// TIA Portal project "EqualAging" (V15)

(* hardware
DEVICE "S7-1200 station_1"  S7-1200 Station
   slot 0: "Rack_0"  S7-1200 Rack  Rack  V1.0
   slot 1: "PLC_1"  CPU 1214C DC/DC/DC  6ES7 214-1AG40-0XB0  V4.2
*)

// ===== PLC "PLC_1"  CPU 1214C DC/DC/DC =====

VAR_GLOBAL   // PLC tag table "Default tag table"
   "Tag_2" AT %Q0.0 : Bool;
   "Tag_3" AT %M1.0 : Bool;
   "Tag_4" AT %M1.1 : Bool;
   "Tag_5" AT %M1.2 : Bool;
   "Tag_6" AT %M1.3 : Bool;
   "Tag_7" AT %M1.4 : Bool;
   "Tag_8" AT %M1.5 : Bool;
   "Tag_9" AT %M1.6 : Bool;
   "Tag_10" AT %MW20 : Int;
   "Tag_11" AT %MD10 : Time;
   "Tag_12" AT %MD11 : Time;
   "Tag_13" AT %MD16 : Time;
   "Clock_Byte" AT %MB0 : Byte;
   "Clock_10Hz" AT %M0.0 : Bool;
   "Clock_5Hz" AT %M0.1 : Bool;
   "Clock_2.5Hz" AT %M0.2 : Bool;
   "Clock_2Hz" AT %M0.3 : Bool;
   "Clock_1.25Hz" AT %M0.4 : Bool;
   "Clock_1Hz" AT %M0.5 : Bool;
   "Clock_0.625Hz" AT %M0.6 : Bool;
   "Clock_0.5Hz" AT %M0.7 : Bool;
   "Tag_1" AT %M10.0 : Bool;
   "Tag_14" AT %M10.1 : Bool;
   "Tag_15" AT %M10.2 : Bool;
   "Tag_16" AT %M10.3 : Bool;
   "Tag_17" AT %M10.4 : Bool;
END_VAR

DATA_BLOCK "EqualAging_DB"   // DB1
{ S7_Optimized_Access := 'TRUE' }
VERSION : 0.1
// stored: InstanceOfName EqualAging
"EqualAging"
BEGIN
END_DATA_BLOCK

FUNCTION_BLOCK "EqualAging"   // FB1, SCL
{ S7_Optimized_Access := 'TRUE' }
VERSION : 0.1
   VAR_INPUT
      i_SystemEnable : Bool;   // Sistemi genel aç/kapat anahtarı
      i_ResetAlarms : Bool;   // Arıza ve saatleri resetler
      i_Clock_1Hz : Bool;   // Saat sayımı için 1 saniyelik darbe
      i_SetMotorCount : Int;   // Çalıştırılmak istenen motor sayısı
      i_StageDelayTime : Time;   // Motorlar arası devreye girme süresi
      i_RotationInterval : Time;   // Motor değişim süresi
      i_M1_Ready : Bool;   // 1. motor hazır/sağlam
      i_M2_Ready : Bool;   // 2. motor hazır/sağlam
      i_M3_Ready : Bool;   // 3. motor hazır/sağlam
      i_M4_Ready : Bool;   // 4. motor hazır/sağlam
      i_M5_Ready : Bool;   // 5. motor hazır/sağlam
   END_VAR
   VAR_OUTPUT
      q_M1_Start : Bool;   // 1. motor çalıştır komutu
      q_M2_Start : Bool;   // 2. motor çalıştır komutu
      q_M3_Start : Bool;   // 3. motor çalıştır komutu
      q_M4_Start : Bool;   // 4. motor çalıştır komutu
      q_M5_Start : Bool;   // 5. motor çalıştır komutu
      q_M1_Hours : Real;   // 1. motor çalışma saati
      q_M2_Hours : Real;   // 2. motor çalışma saati
      q_M3_Hours : Real;   // 3. motor çalışma saati
      q_M4_Hours : Real;   // 4. motor çalışma saati
      q_M5_Hours : Real;   // 5. motor çalışma saati
      q_ActiveCount : Int;   // aktif çalışan motor sayısı
      q_RotationTrigger : Bool;
      q_InsufficientCap : Bool;   // Kapasite yetersiz uyarısı
   END_VAR
   VAR
      stat_RTrig : R_TRIG;   // Saat darbesini yakalamak için
   END_VAR
   VAR RETAIN
      stat_RunSecs : Array[0..5] of DInt;   // motorların toplam süresi
   END_VAR
   VAR
      stat_RotationTimer : TON_TIME;
      stat_CmdStart : Array[0..5] of Bool;   // Çıkışları yönetmek için iç hafıza
      stat_StageTimer : TON_TIME;
   END_VAR
   VAR_TEMP
      temp_i : Int;
      temp_k : Int;
      temp_AvailQty : Int;
      temp_RunQty_1 : Int;
      temp_MinTime : DInt;
      temp_MaxTime : DInt;
      temp_BestStart : Int;
      temp_BestStop : Int;
      temp_Ready : Array[0..5] of Bool;
      temp_SafeSet : Int;
      temp_RunQty : Int;
   END_VAR
BEGIN


   // 1. GİRİŞLERİ DİZİYE AKTARMA (MAPPING)
   #temp_Ready[1] := #i_M1_Ready;
   #temp_Ready[2] := #i_M2_Ready;
   #temp_Ready[3] := #i_M3_Ready;
   #temp_Ready[4] := #i_M4_Ready;
   #temp_Ready[5] := #i_M5_Ready;

   // Saat Palsini Yakala
   #stat_RTrig(CLK := #i_Clock_1Hz);

   #temp_AvailQty := 0;
   #temp_RunQty := 0;

   FOR #temp_i := 1 TO 5 DO
       // Saat Sayacı 
       IF #stat_CmdStart[#temp_i] AND #stat_RTrig.Q THEN
           #stat_RunSecs[#temp_i] := #stat_RunSecs[#temp_i] + 1;
       END_IF;

       // Reset İşlemi 
       IF #i_ResetAlarms THEN
           #stat_RunSecs[#temp_i] := 0;
       END_IF;

       // Hazır Değilse Start'ı Kes
       IF NOT #temp_Ready[#temp_i] THEN
           #stat_CmdStart[#temp_i] := FALSE;
       ELSE
           // Hazırsa "Sağlam" sayısına ekle
           #temp_AvailQty := #temp_AvailQty + 1;
       END_IF;

       // Çalışanları Say 
       IF #stat_CmdStart[#temp_i] THEN
           #temp_RunQty := #temp_RunQty + 1;
       END_IF;
   END_FOR;

   // Çıkışa Aktar
   #q_ActiveCount := #temp_RunQty;

   // Kapasite Kontrolü
   IF #i_SetMotorCount > #temp_AvailQty THEN
       #q_InsufficientCap := TRUE;
       #temp_SafeSet := #temp_AvailQty;
   ELSE
       #q_InsufficientCap := FALSE;
       #temp_SafeSet := #i_SetMotorCount;
   END_IF;

   // --- ROTASYON ZAMANLAYICISI ---
   #stat_RotationTimer(IN := #i_SystemEnable AND
                       (#temp_RunQty = #temp_SafeSet) AND
                       (#temp_RunQty > 0) AND
                       (#temp_AvailQty > #temp_SafeSet),
                       PT := #i_RotationInterval);

   #q_RotationTrigger := #stat_RotationTimer.Q;

   IF #stat_RotationTimer.Q THEN
       #temp_MaxTime := -1;
       #temp_BestStop := 0;

       FOR #temp_k := 1 TO 5 DO
           IF #stat_CmdStart[#temp_k] THEN
               IF #stat_RunSecs[#temp_k] > #temp_MaxTime THEN
                   #temp_MaxTime := #stat_RunSecs[#temp_k];
                   #temp_BestStop := #temp_k;
               END_IF;
           END_IF;
       END_FOR;

       IF #temp_BestStop > 0 THEN
           #stat_CmdStart[#temp_BestStop] := FALSE;
       END_IF;
   END_IF;

   // --- GEÇİŞ ZAMANLAYICISI ---
   #stat_StageTimer(IN := (#temp_RunQty <> #temp_SafeSet) AND #i_SystemEnable,
                    PT := #i_StageDelayTime);

   IF #stat_StageTimer.Q AND #i_SystemEnable THEN

       // START VERME 
       IF #temp_RunQty < #temp_SafeSet THEN
           #temp_MinTime := 2147483647;
           #temp_BestStart := 0;

           FOR #temp_k := 1 TO 5 DO
               IF #temp_Ready[#temp_k] AND NOT #stat_CmdStart[#temp_k] THEN
                   IF #stat_RunSecs[#temp_k] < #temp_MinTime THEN
                       #temp_MinTime := #stat_RunSecs[#temp_k];
                       #temp_BestStart := #temp_k;
                   END_IF;
               END_IF;
           END_FOR;

           IF #temp_BestStart > 0 THEN
               #stat_CmdStart[#temp_BestStart] := TRUE;
           END_IF;

           // STOP VERME
       ELSIF #temp_RunQty > #temp_SafeSet THEN
           #temp_MaxTime := -1;
           #temp_BestStop := 0;

           FOR #temp_k := 1 TO 5 DO
               IF #stat_CmdStart[#temp_k] THEN
                   IF #stat_RunSecs[#temp_k] > #temp_MaxTime THEN
                       #temp_MaxTime := #stat_RunSecs[#temp_k];
                       #temp_BestStop := #temp_k;
                   END_IF;
               END_IF;
           END_FOR;

           IF #temp_BestStop > 0 THEN
               #stat_CmdStart[#temp_BestStop] := FALSE;
           END_IF;
       END_IF;
   END_IF;

   // Sistem Kapalıysa Hepsini Kes
   IF NOT #i_SystemEnable THEN
       FOR #temp_i := 1 TO 5 DO
           #stat_CmdStart[#temp_i] := FALSE;
       END_FOR;
   END_IF;

   // ÇIKIŞLARI AKTARMA
   #q_M1_Start := #stat_CmdStart[1];
   #q_M2_Start := #stat_CmdStart[2];
   #q_M3_Start := #stat_CmdStart[3];
   #q_M4_Start := #stat_CmdStart[4];
   #q_M5_Start := #stat_CmdStart[5];

   #q_M1_Hours := DINT_TO_REAL(#stat_RunSecs[1]) / 3600.0;
   #q_M2_Hours := DINT_TO_REAL(#stat_RunSecs[2]) / 3600.0;
   #q_M3_Hours := DINT_TO_REAL(#stat_RunSecs[3]) / 3600.0;
   #q_M4_Hours := DINT_TO_REAL(#stat_RunSecs[4]) / 3600.0;
   #q_M5_Hours := DINT_TO_REAL(#stat_RunSecs[5]) / 3600.0;
END_FUNCTION_BLOCK

ORGANIZATION_BLOCK "Main"   // OB1, LAD, ProgramCycle
TITLE = "Main Program Sweep (Cycle)"
{ S7_Optimized_Access := 'TRUE' }
VERSION : 0.1
   VAR_INPUT
      Initial_Call : Bool;   // Initial call of this OB
      Remanence : Bool;   // =True, if remanent data are available
   END_VAR
BEGIN

REGION Network 1
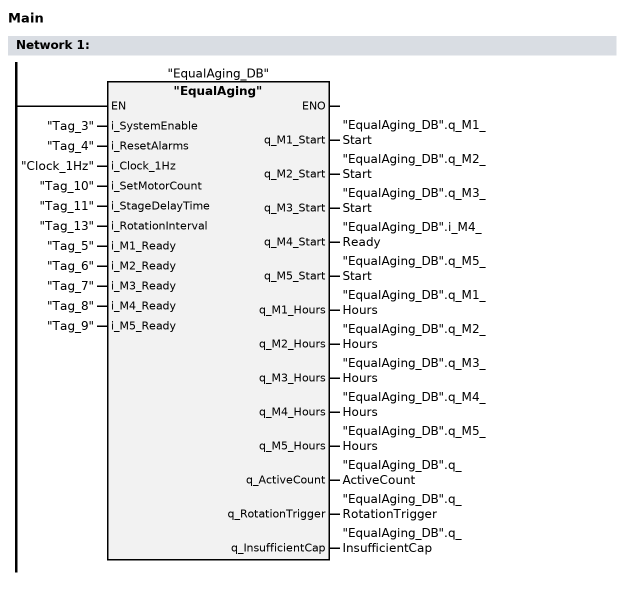
   RUNG wire#powerrail
      "EqualAging_DB"(i_SystemEnable := "Tag_3", i_ResetAlarms := "Tag_4", i_Clock_1Hz := "Clock_1Hz", i_SetMotorCount := "Tag_10", i_StageDelayTime := "Tag_11", i_RotationInterval := "Tag_13", i_M1_Ready := "Tag_5", i_M2_Ready := "Tag_6", i_M3_Ready := "Tag_7", i_M4_Ready := "Tag_8", i_M5_Ready := "Tag_9", q_M1_Start => "EqualAging_DB".q_M1_Start, q_M2_Start => "EqualAging_DB".q_M2_Start, q_M3_Start => "EqualAging_DB".q_M3_Start, q_M4_Start => "EqualAging_DB".i_M4_Ready, q_M5_Start => "EqualAging_DB".q_M5_Start, q_M1_Hours => "EqualAging_DB".q_M1_Hours, q_M2_Hours => "EqualAging_DB".q_M2_Hours, q_M3_Hours => "EqualAging_DB".q_M3_Hours, q_M4_Hours => "EqualAging_DB".q_M4_Hours, q_M5_Hours => "EqualAging_DB".q_M5_Hours, q_ActiveCount => "EqualAging_DB".q_ActiveCount, q_RotationTrigger => "EqualAging_DB".q_RotationTrigger, q_InsufficientCap => "EqualAging_DB".q_InsufficientCap)
   END_RUNG
   // the same network as SCL:
   "EqualAging_DB"(i_SystemEnable := "Tag_3",   // "EqualAging"
                   i_ResetAlarms := "Tag_4",
                   i_Clock_1Hz := "Clock_1Hz",
                   i_SetMotorCount := "Tag_10",
                   i_StageDelayTime := "Tag_11",
                   i_RotationInterval := "Tag_13",
                   i_M1_Ready := "Tag_5",
                   i_M2_Ready := "Tag_6",
                   i_M3_Ready := "Tag_7",
                   i_M4_Ready := "Tag_8",
                   i_M5_Ready := "Tag_9",
                   q_M1_Start => "EqualAging_DB".q_M1_Start,
                   q_M2_Start => "EqualAging_DB".q_M2_Start,
                   q_M3_Start => "EqualAging_DB".q_M3_Start,
                   q_M4_Start => "EqualAging_DB".i_M4_Ready,
                   q_M5_Start => "EqualAging_DB".q_M5_Start,
                   q_M1_Hours => "EqualAging_DB".q_M1_Hours,
                   q_M2_Hours => "EqualAging_DB".q_M2_Hours,
                   q_M3_Hours => "EqualAging_DB".q_M3_Hours,
                   q_M4_Hours => "EqualAging_DB".q_M4_Hours,
                   q_M5_Hours => "EqualAging_DB".q_M5_Hours,
                   q_ActiveCount => "EqualAging_DB".q_ActiveCount,
                   q_RotationTrigger => "EqualAging_DB".q_RotationTrigger,
                   q_InsufficientCap => "EqualAging_DB".q_InsufficientCap);
END_REGION
END_ORGANIZATION_BLOCK